(* IEC 61131-3 sources: exOS-Demos/NodeRed/Components/Source/SimPanel/SimPanel, 2 files *)

(* ---- SimPanel.typ ---- *)
TYPE
	SimPanelKnobs : 	STRUCT
		P1 : INT;
		P2 : INT;
	END_STRUCT;
	SimPanelSwitches : 	STRUCT
		DI1 : BOOL;
		DI2 : BOOL;
	END_STRUCT;
	SimPanelLED : 	STRUCT
		Green : BOOL;
		Red : BOOL;
		Yellow : BOOL;
	END_STRUCT;
	SimPanelLEDs : 	STRUCT
		DI1 : BOOL;
		DI2 : BOOL;
		DI3 : SimPanelLED;
		DI4 : SimPanelLED;
		DI5 : SimPanelLED;
		DI6 : SimPanelLED;
	END_STRUCT;
	SimPanelButtons : 	STRUCT
		DI3 : BOOL;
		DI4 : BOOL;
		DI5 : BOOL;
		DI6 : BOOL;
		Encoder : BOOL;
	END_STRUCT;
	SimPanel : 	STRUCT
		Switches : SimPanelSwitches; (*PUB*)
		Buttons : SimPanelButtons; (*PUB*)
		LEDs : SimPanelLEDs; (*SUB*)
		Knobs : SimPanelKnobs; (*PUB*)
		Display : INT; (*SUB*)
		Encoder : UINT; (*PUB*)
	END_STRUCT;
END_TYPE

(* ---- SimPanel.fun ---- *)
FUNCTION_BLOCK SimPanelInit
	VAR_OUTPUT
		Handle : UDINT;
	END_VAR
	VAR
		_state : USINT;
	END_VAR
END_FUNCTION_BLOCK

FUNCTION_BLOCK SimPanelCyclic
	VAR_INPUT
		Enable : BOOL;
		Handle : UDINT;
		Start : BOOL;
		pSimPanel : REFERENCE TO SimPanel;
	END_VAR
	VAR_OUTPUT
		Active : BOOL;
		Error : BOOL;
		Disconnected : BOOL;
		Connected : BOOL;
		Operational : BOOL;
		Aborted : BOOL;
	END_VAR
	VAR
		_state : USINT;
	END_VAR
END_FUNCTION_BLOCK

FUNCTION_BLOCK SimPanelExit
	VAR_INPUT
		Handle : UDINT;
	END_VAR
	VAR
		_state : USINT;
	END_VAR
END_FUNCTION_BLOCK
